FUNCTION_BLOCK ExampleCylinderMoveTask EXTENDS TcoCore.TcoTask
VAR_INPUT
    PositionSensor         : BOOL;
    MaxTimeToReachPosition : TIME := T#10S;
    PositionName           : STRING(25);
END_VAR
VAR_IN_OUT
    MoveToPositionSignal : BOOL;
    InverseSignal        : BOOL;
END_VAR

VAR
    _stringBuilder : TcoCore.StringBuilder;
END_VAR

IF (THIS^.Execute()) THEN
    IF (THIS^.ElapsedTime > MaxTimeToReachPosition) THEN
        THIS^.Messenger
            .Warning(_stringBuilder.Clear().Append(PositionName).Append(' sensor not reached yet.').ToString());
    END_IF;

    InverseSignal        := FALSE;
    MoveToPositionSignal := TRUE;
    THIS^.DoneWhen(PositionSensor);
END_IF

METHOD PUBLIC FB_init : BOOL
VAR_INPUT
    bInitRetains : BOOL; // if TRUE, the retain variables are initialized (warm start / cold start)
    bInCopyCode  : BOOL; // if TRUE, the instance afterwards gets moved into the copy code (online change)
    ParentObject : ITcoObject;
END_VAR
END_METHOD

(*~
    <docu>
        <summary>
            Executes when task is aborted.
        </summary>
    </docu>
~*)
METHOD PROTECTED OnAbort
MoveToPositionSignal := FALSE;
END_METHOD

METHOD PROTECTED OnError
END_METHOD

END_FUNCTION_BLOCK

(* stored: Version 1.1.0.1, ProductVersion 3.1.4024.12
   POU ExampleCylinderMoveTask: Id {a246bb94-06eb-46db-ac8a-d49f03e8b61b}, SpecialFunc None
   Method FB_init: Id {bfbf43ca-b77c-4e1e-9b19-251c8724464e}
   Method OnAbort: Id {e9f5c521-7aac-466a-bc99-32ae6f7b22db}
   Method OnError: Id {089bfd42-5b8c-405d-a704-8e081af9ad5c} *)
